// TIA Portal V18 export
// export: Created 2026-06-12T02:00:00Z, ExportSetting WithDefaults
VAR_GLOBAL   // PLC tag table "PLC_AI_B6_Tags"
   AI_B6_TICR211_Temp AT %MD600 : Real;   // TEMP 50-80 °C
   AI_B6_TICR210_Temp AT %MD604 : Real;   // TEMP 50-80 °C
   AI_B6_TICR201_Tank_Temp AT %MD608 : Real;   // TEMP 50-80 °C
   AI_B6_PT201_Pressure AT %MD612 : Real;   // PRESSURE 7-8 bar
   AI_B6_Ph201_pH AT %MD616 : Real;   // COUNT 6-8 pH
   AI_B6_ORP201_ORP AT %MD620 : Real;   // COUNT 20-80 %
   AI_B6_DPL101_Level AT %MD624 : Real;   // LEVEL 100-500 L
   AI_B6_TICR214_Temp AT %MD628 : Real;   // TEMP 50-80 °C
   AI_B6_TICR204_Temp AT %MD632 : Real;   // TEMP 50-80 °C
   AI_B6_TICR205_Temp AT %MD636 : Real;   // TEMP 50-80 °C
   AI_B6_TICR206_Temp AT %MD640 : Real;   // TEMP 50-80 °C
   AI_B6_FHC203_Flow AT %MD644 : Real;   // FLOW 100-200 L/h
   AI_B6_BPC201_Pressure AT %MD648 : Real;   // PRESSURE 7-8 bar
END_VAR
